(* CoDeSys 2.3 export: EV_DOBLE.EXP *)

(* Data type *)
TYPE EV_Doble :
STRUCT
	Activa_Mas     : BOOL;
      Activa_Menos  : BOOL;
END_STRUCT
END_TYPE
